// TwinCAT 3 PLC project AngerbauerWilhelm
// ProgramVersion: 3.1.4023.0
// libraries:
//   EfficientIO Communicator, * (EfficientIO)
//   EfficientIO Energy Basic, * (EfficientIO)
//   EfficientIO ModbusTCP, * (EfficientIO)
//   Lynus Persistent Data V1, * (Lynus AG)
//   Lynus Standards, * (EfficientIO)
//   Tc2_Standard, * (Beckhoff Automation GmbH)
//   Tc2_System, * (Beckhoff Automation GmbH)
//   Tc2_TcpIp, * (Beckhoff Automation GmbH)
//   Tc2_Utilities, * (Beckhoff Automation GmbH)
//   Tc3_Module, * (Beckhoff Automation GmbH)
// project tree:
//   / FastTask.TcTTO, PlcTask.TcTTO, SlowTask.TcTTO
//   FBs/ fb_Convert4BytesToLreal.TcPOU (not stored), FB_ModBus_100Registers_FC3.TcPOU, FB_ModBus_2Registers_FC3.TcPOU (not stored), FB_TCPModbusRequest_PV.TcPOU, FB_TCPModbusRequest_Grid.TcPOU
//   POUs/ prgComEffIO.TcPOU, prgGrid.TcPOU, prgPersistent.TcPOU (not stored), prgPV.TcPOU, prgRWEffIO.TcPOU, prgTCP.TcPOU, prgVarEffIO.TcPOU
// real-time tasks:
//   TASK MiddleTask: cycle T#10ms, priority 20, ADS port 350
//   TASK FastTask: cycle T#5ms, priority 19, ADS port 351
//   TASK SlowTask: cycle T#20ms, priority 21, ADS port 352

CONFIGURATION AngerbauerWilhelm
    RESOURCE PLC ON TwinCAT3
        TASK FastTask(INTERVAL := T#5ms, PRIORITY := 19);
        TASK PlcTask(INTERVAL := T#10ms, PRIORITY := 20);
        TASK SlowTask(INTERVAL := T#20ms, PRIORITY := 21);
        PROGRAM prgRWEffIO WITH FastTask : prgRWEffIO;
        PROGRAM prgVarEffIO WITH FastTask : prgVarEffIO;
        PROGRAM prgTCP WITH PlcTask : prgTCP;
        PROGRAM prgPV WITH PlcTask : prgPV;
        PROGRAM prgPersistent WITH PlcTask : prgPersistent;
        PROGRAM prgGrid WITH PlcTask : prgGrid;
        PROGRAM prgComEffIO WITH SlowTask : prgComEffIO;
    END_RESOURCE
END_CONFIGURATION

// ---- POUs/prgRWEffIO.TcPOU
PROGRAM prgRWEffIO
VAR
	fbRW1		: FB_ReadWrite_V2;
END_VAR

fbRW1(eUploadType:=	eSelectDataUploadType.e_Change_Intervall5min, 
					bBusy=> , 
					bError=> , 
					udiErrorCodeOut=> , 
					eErrorReadWrite_Out=> );

END_PROGRAM

// ---- POUs/prgVarEffIO.TcPOU
PROGRAM prgVarEffIO
VAR
	fbVar		: FB_VarInfo;
END_VAR

fbVar(
	bReadInfo:= , 
	eTMCFile:= eSelectTMCFile.eDontUseTMCFile, 
	eSavePositionTMCFile:= eSavePositionOnPLC.ePostionC, 
	udiCounterFoundVariables=> , 
	bError=> , 
	bBusy=> , 
	byProgress=> , 
	udiErrorCodeOut=> , 
	eErrorVarInfo_Out=> , 
	sVarWithError=> );

END_PROGRAM

// ---- POUs/prgTCP.TcPOU
PROGRAM prgTCP
VAR
	FB_SocketConnect : FB_SocketConnect;
	bExecuteSC: BOOL;
	hSocket : T_HSOCKET;
	FB_SocketSend : FB_SocketSend;
	sSendString : STRING(255);
	byteSendString : ARRAY[1..12] OF BYTE;
	bExecuteSS: BOOL;
	FB_SocketReceive : FB_SocketReceive;
	byteReceiveString : ARRAY[1..200] OF BYTE;
	FB_BYTE_TO_WORD : FB_CV_BYTE_TO_WORD;
	FB_WORD_TO_INT : FB_CV_WORD_TO_INT;
	wTemp : WORD;
	iOutput : INT;

END_VAR

FB_SocketConnect(
	sSrvNetId := '',
	sRemoteHost := '10.0.0.4',
	nRemotePort := 502,
	bExecute := bExecuteSC,
	tTimeout := T#1S,
	bBusy =>,
	bError =>,
	nErrId =>,
	hSocket => hSocket);
	
FB_SocketSend(
	sSrvNetId:= '', 
	hSocket:= hSocket, 
	cbLen:= 12,
	pSrc:= ADR( byteSendString ), 
	bExecute:= bExecuteSS, 
	tTimeout:= T#3S, 
	bBusy=> , 
	bError=> , 
	nErrId=> );

FB_SocketReceive(
	sSrvNetId:= '', 
	hSocket:= hSocket, 
	cbLen:= 200, 
	pDest:= ADR( byteReceiveString ), 
	bExecute:= , 
	tTimeout:= T#3S, 
	bBusy=> , 
	bError=> , 
	nErrId=> , 
	nRecBytes=> );
	
FB_BYTE_TO_WORD(byInputValue_1 := byteReceiveString[12],byInputValue_2 := byteReceiveString[13], Ebyteorderforconvert := Ebyteorder.EBIGENDIAN, woutputvalue => wTemp);
FB_WORD_TO_INT(wInputValue := wTemp, iOutputValue => iOutput);

END_PROGRAM

// ---- POUs/prgPV.TcPOU
PROGRAM prgPV
VAR
	fbPVCounter1		: FB_EnergyCounter;
	fbPVCounter2		: FB_EnergyCounter;
	lrPowerPV1			: LREAL;				//{#lynus.ag#()}
	lrPowerPV2			: LREAL;				//{#lynus.ag#()}
	lrPowerPVTotal		: LREAL;				//{#lynus.ag#()}
	byErrorWarningPV	: BYTE;					//{#lynus.ag#()}
	FB_PV1:FB_TCPModbusRequest_PV;
	FB_PV2:FB_TCPModbusRequest_PV;
	lrVoltagePV1_L1L2_V		: LREAL;				//{#lynus.ag#()}
	lrVoltagePV1_L2L3_V		: LREAL;				//{#lynus.ag#()}
	lrVoltagePV1_L3L1_V		: LREAL;				//{#lynus.ag#()}
	lrVoltagePV2_L1L2_V		: LREAL;				//{#lynus.ag#()}
	lrVoltagePV2_L2L3_V		: LREAL;				//{#lynus.ag#()}
	lrVoltagePV2_L3L1_V		: LREAL;				//{#lynus.ag#()}
END_VAR
VAR PERSISTENT
	lrCounterPV1		: LREAL;					//{#lynus.ag#()}
	lrCounterPV2		: LREAL;					//{#lynus.ag#()}
	lrCounterPVTotal	: LREAL;					//{#lynus.ag#()}
END_VAR


FB_PV1	(	b_Enable:= TRUE, 
			str_IPAdress:= '10.0.0.4', 
			lreal_RealPower_kW=> lrPowerPV1,
			lreal_Voltage_L1L2_V=> lrVoltagePV1_L1L2_V , 
			lreal_Voltage_L2L3_V=> lrVoltagePV1_L2L3_V , 
			lreal_Voltage_L3L1_V=> lrVoltagePV1_L3L1_V);


fbPVCounter1(	byActiveTariff := 1,	
				lrPowerInput := 0-lrPowerPV1,
				lrTotalCounterEnergy_Production => lrCounterPV1);
	

FB_PV2	(	b_Enable:= TRUE, 
			str_IPAdress:= '10.0.0.5', 
			lreal_RealPower_kW=> lrPowerPV2,
			lreal_Voltage_L1L2_V=> lrVoltagePV2_L1L2_V , 
			lreal_Voltage_L2L3_V=> lrVoltagePV2_L2L3_V , 
			lreal_Voltage_L3L1_V=> lrVoltagePV2_L3L1_V);

fbPVCounter2(	byActiveTariff := 1,	
				lrPowerInput := 0-lrPowerPV2,
				lrTotalCounterEnergy_Production => lrCounterPV2);
	
lrPowerPVTotal := lrPowerPV1 + lrPowerPV2;
lrCounterPVTotal := lrCounterPV1 + lrCounterPV2;

END_PROGRAM

// ---- FBs/FB_TCPModbusRequest_PV.TcPOU
FUNCTION_BLOCK FB_TCPModbusRequest_PV
VAR_INPUT
	b_Enable: BOOL;
	str_IPAdress: STRING(15);
	
		
END_VAR
VAR_OUTPUT

	lreal_RealPower_kW:LREAL;
	lreal_Voltage_L1L2_V: LREAL;
	lreal_Voltage_L2L3_V: LREAL;
	lreal_Voltage_L3L1_V: LREAL;
	lreal_Voltage_L1_V: LREAL;
	lreal_Voltage_L2_V: LREAL;
	lreal_Voltage_L3_V: LREAL;
	lreal_Current_L1_A: LREAL;
	lreal_Current_L2_A: LREAL;
	lreal_Current_L3_A: LREAL;
	lreal_PeakPowerDay_kW: LREAL;
	lreal_Power2_kW: LREAL;
	lreal_ReactivePower_kVAr: LREAL;
	lreal_PowerFactor: LREAL;
	lreal_Frequency_Hz: LREAL;
	lreal_Efficiency: LREAL;
	lreal_InternalTemperature_C: LREAL;
	lreal_IsolationResistance_MOhm: LREAL;
END_VAR
VAR
	i_State:INT;
	FB_SocketConnect : FB_SocketConnect;
	hSocket : T_HSOCKET;
	FB_SocketSend : FB_SocketSend;
	FB_SocketReceive : FB_SocketReceive;
	byteSendString : ARRAY[1..12] OF BYTE;
	FB_CloseSockets: FB_SocketCloseAll;
	
	ton_TimeOut: Ton;
	ton_WaitforReconnect: Ton;
	ton_ConnectionEstablised: Ton;
	time_ReconnectTime:TIME:=T#30M;
	b_configured: BOOL;
	byteReceiveString : ARRAY[1..200] OF BYTE;
	FB_BYTE_TO_WORD_1 : FB_CV_BYTE_TO_WORD;
	FB_BYTE_TO_WORD_2 : FB_CV_BYTE_TO_WORD;
	FB_WORD_TO_INT : FB_CV_WORD_TO_INT;
	ton_WaitforNetxtRequest: Ton;
	ton_Wait: Ton;
	int_SuccessCounter: INT;
	int_ReconnectCounter: INT;
	int_ErrorCount: INT;
	fbConvertWordToDword		: FB_CV_WORD_TO_DWORD;			//Convert Word to Dword
	fb_ConvertBytesToLreal		:fb_Convert4BytesToLreal;

END_VAR





IF NOT b_Enable THEN			// go to state 0 if not enabled
	i_State := 0;
END_IF


CASE i_State OF
	0:	// wait for enable state
		IF b_Enable THEN
			i_State := 1;
		END_IF
		FB_SocketConnect.bExecute := FALSE;
		FB_SocketSend.bExecute := FALSE;
		FB_SocketSend.bExecute := FALSE;
		ton_TimeOut.IN :=FALSE;	
		ton_ConnectionEstablised.IN := FALSE;
	

	1: // check if configured
		IF b_configured = FALSE THEN
			// request FC3, Register 32064, 25 Words --> Real PV Power ff
			byteSendString[1] := 0;
			byteSendString[2] := 1;
			byteSendString[3] := 0;
			byteSendString[4] := 0;
			byteSendString[5] := 0;
			byteSendString[6] := 6;
			byteSendString[7] := 1;
			byteSendString[8] := 3;
			byteSendString[9] := 125;
			byteSendString[10] := 64;
			byteSendString[11] := 0;
			byteSendString[12] := 25;
		
			b_configured := TRUE;
		END_IF
		i_State := i_State+1;
		
	2: // open socket
		FB_SocketConnect.bExecute := TRUE;
		ton_TimeOut.IN :=TRUE;
		i_State := i_State+1;
		
	3: // wait for connection established	
		IF NOT FB_SocketConnect.bBusy AND NOT FB_SocketConnect.bError THEN
			ton_TimeOut.IN :=FALSE;
			ton_ConnectionEstablised.IN := TRUE;
			i_State := i_State+1;
		ELSIF FB_SocketConnect.bError OR ton_TimeOut.Q THEN
			ton_TimeOut.IN :=FALSE;
			i_State := 100;
		END_IF
	
	4: //connection established, request data
		ton_Wait.IN := TRUE;
		IF ton_Wait.Q THEN
			FB_SocketSend.bExecute := TRUE;
			ton_TimeOut.IN :=TRUE;
			ton_Wait.IN := FALSE;
			i_State := i_State+1;
		END_IF
	
	5: // wait for request sent
		IF NOT FB_SocketSend.bBusy AND NOT FB_SocketSend.bError THEN
			ton_TimeOut.IN :=FALSE;
			FB_SocketSend.bExecute := FALSE;
			i_State := i_State+1;  
		ELSIF FB_SocketSend.bError OR ton_TimeOut.Q THEN
			FB_SocketSend.bExecute := FALSE;
			ton_TimeOut.IN :=FALSE;
			i_State := 100;
		END_IF
		
	6: // wait for data
		ton_Wait.IN := TRUE;
		IF ton_Wait.Q THEN
			FB_SocketReceive.bExecute := TRUE;
			ton_Wait.IN := FALSE;
			i_State := i_State+1; 
		END_IF		 
	
	7:	
		ton_Wait.IN := TRUE;
		IF ton_Wait.Q THEN
			ton_TimeOut.IN :=TRUE;
			i_State := i_State+1; 
		END_IF	
	
	8: // convert received data
		IF NOT FB_SocketReceive.bBusy AND NOT FB_SocketReceive.bError THEN
			int_SuccessCounter := int_SuccessCounter+1;
			ton_TimeOut.IN :=FALSE;
			FB_SocketReceive.bExecute := FALSE;
	
			FB_BYTE_TO_WORD_1(byInputValue_1 := byteReceiveString[14],byInputValue_2 := byteReceiveString[15], Ebyteorderforconvert := Ebyteorder.EBIGENDIAN, woutputvalue => );
			lreal_Voltage_L1L2_V := WORD_TO_LREAL(FB_BYTE_TO_WORD_1.woutputvalue)/10;
			FB_BYTE_TO_WORD_1(byInputValue_1 := byteReceiveString[16],byInputValue_2 := byteReceiveString[17], Ebyteorderforconvert := Ebyteorder.EBIGENDIAN, woutputvalue => );
			lreal_Voltage_L2L3_V := WORD_TO_LREAL(FB_BYTE_TO_WORD_1.woutputvalue)/10;
			FB_BYTE_TO_WORD_1(byInputValue_1 := byteReceiveString[18],byInputValue_2 := byteReceiveString[19], Ebyteorderforconvert := Ebyteorder.EBIGENDIAN, woutputvalue => );
			lreal_Voltage_L3L1_V := WORD_TO_LREAL(FB_BYTE_TO_WORD_1.woutputvalue)/10;
			FB_BYTE_TO_WORD_1(byInputValue_1 := byteReceiveString[20],byInputValue_2 := byteReceiveString[21], Ebyteorderforconvert := Ebyteorder.EBIGENDIAN, woutputvalue => );
			lreal_Voltage_L1_V := WORD_TO_LREAL(FB_BYTE_TO_WORD_1.woutputvalue)/10;
			FB_BYTE_TO_WORD_1(byInputValue_1 := byteReceiveString[22],byInputValue_2 := byteReceiveString[23], Ebyteorderforconvert := Ebyteorder.EBIGENDIAN, woutputvalue => );
			lreal_Voltage_L2_V := WORD_TO_LREAL(FB_BYTE_TO_WORD_1.woutputvalue)/10;
			FB_BYTE_TO_WORD_1(byInputValue_1 := byteReceiveString[24],byInputValue_2 := byteReceiveString[25], Ebyteorderforconvert := Ebyteorder.EBIGENDIAN, woutputvalue => );
			lreal_Voltage_L3_V := WORD_TO_LREAL(FB_BYTE_TO_WORD_1.woutputvalue)/10;


			fb_ConvertBytesToLreal(	by_InputValue_1:= byteReceiveString[10], 
									by_InputValue_2:= byteReceiveString[11], 
									by_InputValue_3:= byteReceiveString[12], 
									by_InputValue_4:= byteReceiveString[13], 
									int_Divider:= 1000, 
									lreal_Output=> );

			IF fb_ConvertBytesToLreal.lreal_Output < 30 AND fb_ConvertBytesToLreal.lreal_Output > -1 THEN
				lreal_RealPower_kW := fb_ConvertBytesToLreal.lreal_Output;
			END_IF
			
			fb_ConvertBytesToLreal(	by_InputValue_1:= byteReceiveString[26], 
									by_InputValue_2:= byteReceiveString[27], 
									by_InputValue_3:= byteReceiveString[28], 
									by_InputValue_4:= byteReceiveString[29], 
									int_Divider:= 1000, 
									lreal_Output=> lreal_Current_L1_A);
									
			fb_ConvertBytesToLreal(	by_InputValue_1:= byteReceiveString[30], 
									by_InputValue_2:= byteReceiveString[31], 
									by_InputValue_3:= byteReceiveString[32], 
									by_InputValue_4:= byteReceiveString[33], 
									int_Divider:= 1000, 
									lreal_Output=> lreal_Current_L2_A);

			fb_ConvertBytesToLreal(	by_InputValue_1:= byteReceiveString[34], 
									by_InputValue_2:= byteReceiveString[35], 
									by_InputValue_3:= byteReceiveString[36], 
									by_InputValue_4:= byteReceiveString[37], 
									int_Divider:= 1000, 
									lreal_Output=> lreal_Current_L3_A);
									
			fb_ConvertBytesToLreal(	by_InputValue_1:= byteReceiveString[38], 
									by_InputValue_2:= byteReceiveString[39], 
									by_InputValue_3:= byteReceiveString[40], 
									by_InputValue_4:= byteReceiveString[41], 
									int_Divider:= 1000, 
									lreal_Output=> lreal_PeakPowerDay_kW );

			fb_ConvertBytesToLreal(	by_InputValue_1:= byteReceiveString[42], 
									by_InputValue_2:= byteReceiveString[43], 
									by_InputValue_3:= byteReceiveString[44], 
									by_InputValue_4:= byteReceiveString[45], 
									int_Divider:= 1000, 
									lreal_Output=> lreal_Power2_kW);
			
			fb_ConvertBytesToLreal(	by_InputValue_1:= byteReceiveString[46], 
									by_InputValue_2:= byteReceiveString[47], 
									by_InputValue_3:= byteReceiveString[48], 
									by_InputValue_4:= byteReceiveString[49], 
									int_Divider:= 1000, 
									lreal_Output=>lreal_ReactivePower_kVAr );

			FB_BYTE_TO_WORD_1(byInputValue_1 := byteReceiveString[50],byInputValue_2 := byteReceiveString[51], Ebyteorderforconvert := Ebyteorder.EBIGENDIAN, woutputvalue => );
			lreal_PowerFactor := WORD_TO_LREAL(FB_BYTE_TO_WORD_1.woutputvalue)/1000;
			FB_BYTE_TO_WORD_1(byInputValue_1 := byteReceiveString[52],byInputValue_2 := byteReceiveString[53], Ebyteorderforconvert := Ebyteorder.EBIGENDIAN, woutputvalue => );
			lreal_Frequency_Hz := WORD_TO_LREAL(FB_BYTE_TO_WORD_1.woutputvalue)/100;
			FB_BYTE_TO_WORD_1(byInputValue_1 := byteReceiveString[54],byInputValue_2 := byteReceiveString[55], Ebyteorderforconvert := Ebyteorder.EBIGENDIAN, woutputvalue => );
			lreal_Efficiency := WORD_TO_LREAL(FB_BYTE_TO_WORD_1.woutputvalue)/100;
			FB_BYTE_TO_WORD_1(byInputValue_1 := byteReceiveString[56],byInputValue_2 := byteReceiveString[57], Ebyteorderforconvert := Ebyteorder.EBIGENDIAN, woutputvalue => );
			lreal_InternalTemperature_C := WORD_TO_LREAL(FB_BYTE_TO_WORD_1.woutputvalue)/10;
			FB_BYTE_TO_WORD_1(byInputValue_1 := byteReceiveString[58],byInputValue_2 := byteReceiveString[59], Ebyteorderforconvert := Ebyteorder.EBIGENDIAN, woutputvalue => );
			lreal_IsolationResistance_MOhm := WORD_TO_LREAL(FB_BYTE_TO_WORD_1.woutputvalue)/1000;

		
			//FB_WORD_TO_INT(wInputValue := FB_BYTE_TO_WORD.woutputvalue, iOutputValue => );
			//lreal_RealPower_kW := (INT_TO_LREAL(FB_WORD_TO_INT.iOutputValue))/1000;

			i_State := i_State+1;
		ELSIF FB_SocketSend.bError OR ton_TimeOut.Q THEN
 			FB_SocketReceive.bExecute := FALSE;
			ton_TimeOut.IN :=FALSE;
			i_State := 100;
		END_IF
	
	9: // for for next request
		ton_WaitforNetxtRequest.IN := TRUE;
		IF NOT b_Enable THEN
			ton_WaitforNetxtRequest.IN := FALSE;
			i_State := 10;
		END_IF
		IF ton_WaitforNetxtRequest.Q THEN
			ton_WaitforNetxtRequest.IN := FALSE;
			i_State := 4;
		END_IF
		IF 	ton_ConnectionEstablised.Q THEN 
			ton_WaitforNetxtRequest.IN := FALSE;
			i_State := 10;
		END_IF

	10: // close sockets
		FB_CloseSockets.bExecute := TRUE;
		ton_TimeOut.IN :=TRUE;
		i_State := i_State+1;
		
	11: // wait for sockets closed
		
		IF NOT FB_CloseSockets.bBusy THEN
			int_ReconnectCounter := int_ReconnectCounter+1;
			FB_CloseSockets.bExecute := FALSE;
			i_State := 0;
		ELSIF FB_CloseSockets.bError THEN
			int_ReconnectCounter := int_ReconnectCounter+1;
			FB_CloseSockets.bExecute := FALSE;
			i_State := 0;
		END_IF

	100: // wait state for reconect
		
		FB_SocketConnect.bExecute := FALSE;
		FB_SocketSend.bExecute := FALSE;
		FB_SocketReceive.bExecute := FALSE;
		ton_ConnectionEstablised.IN := FALSE;
		ton_TimeOut.IN :=FALSE;
		ton_WaitforReconnect.IN := TRUE;
		IF ton_WaitforReconnect.Q THEN
			int_ErrorCount := int_ErrorCount+1;
			ton_WaitforReconnect.IN := FALSE;
			i_State := 10;
		END_IF
	
END_CASE



FB_SocketConnect(
	sSrvNetId := '',
	sRemoteHost := str_IPAdress,
	nRemotePort := 502,
	bExecute := ,
	tTimeout := T#1S,
	bBusy =>,
	bError =>,
	nErrId =>,
	hSocket => hSocket);
	
FB_SocketSend(
	sSrvNetId:= '', 
	hSocket:= hSocket, 
	cbLen:= 12,
	pSrc:= ADR( byteSendString ), 
	bExecute:= , 
	tTimeout:= T#3S, 
	bBusy=> , 
	bError=> , 
	nErrId=> );
	
FB_SocketReceive(
	sSrvNetId:= '', 
	hSocket:= hSocket, 
	cbLen:= 200, 
	pDest:= ADR( byteReceiveString ), 
	bExecute:= , 
	tTimeout:= T#3S, 
	bBusy=> , 
	bError=> , 
	nErrId=> , 
	nRecBytes=> );

FB_CloseSockets(
	sSrvNetId:= '', 
	bExecute:= , 
	tTimeout:= T#2S, 
	bBusy=> , 
	bError=> , 
	nErrId=> );
	
ton_TimeOut(PT := T#5S);
ton_WaitforReconnect(PT := T#10S);
ton_ConnectionEstablised(pt := time_ReconnectTime);
ton_WaitforNetxtRequest(PT:= T#10S);
ton_Wait(PT:=T#2S);

END_FUNCTION_BLOCK

// ---- POUs/prgGrid.TcPOU
PROGRAM prgGrid
VAR
	FB_PV1:FB_TCPModbusRequest_Grid;
	FB_PV2:FB_TCPModbusRequest_Grid;

	lreal_GridVoltage_L1L2_V_PV1		: LREAL;				//{#lynus.ag#()}
	lreal_GridVoltage_L2L3_V_PV1		: LREAL;				//{#lynus.ag#()}
	lreal_GridVoltage_L3L1_V_PV1		: LREAL;				//{#lynus.ag#()}
	lreal_GridVoltage_L1_V_PV1			: LREAL;				//{#lynus.ag#()}
	lreal_GridVoltage_L2_V_PV1			: LREAL;				//{#lynus.ag#()}
	lreal_GridVoltage_L3_V_PV1			: LREAL;				//{#lynus.ag#()}
	lreal_GridCurrent_L1_A_PV1			: LREAL;				//{#lynus.ag#()}
	lreal_GridCurrent_L2_A_PV1			: LREAL;				//{#lynus.ag#()}
	lreal_GridCurrent_L3_A_PV1			: LREAL;				//{#lynus.ag#()}
	lreal_GridPower_kW_PV1				: LREAL;				//{#lynus.ag#()}
	lreal_GridPower_kW_PV1_2			: LREAL;				//{#lynus.ag#()}
	lreal_GridReactivePower_kVAr_PV1	: LREAL;				//{#lynus.ag#()}
	lreal_GridPowerFactor_PV1			: LREAL;				//{#lynus.ag#()}
	lreal_GridFrequency_Hz_PV1			: LREAL;				//{#lynus.ag#()}
	lreal_GridEnergyDelivered_kWh_PV1	: LREAL;				//{#lynus.ag#()}
	lreal_GridEnergySupllied_kWh_PV1	: LREAL;				//{#lynus.ag#()}
	
	lreal_GridVoltage_L1L2_V_PV2		: LREAL;				//{#lynus.ag#()}
	lreal_GridVoltage_L2L3_V_PV2		: LREAL;				//{#lynus.ag#()}
	lreal_GridVoltage_L3L1_V_PV2		: LREAL;				//{#lynus.ag#()}
	lreal_GridVoltage_L1_V_PV2			: LREAL;				//{#lynus.ag#()}
	lreal_GridVoltage_L2_V_PV2			: LREAL;				//{#lynus.ag#()}
	lreal_GridVoltage_L3_V_PV2			: LREAL;				//{#lynus.ag#()}
	lreal_GridCurrent_L1_A_PV2			: LREAL;				//{#lynus.ag#()}
	lreal_GridCurrent_L2_A_PV2			: LREAL;				//{#lynus.ag#()}
	lreal_GridCurrent_L3_A_PV2			: LREAL;				//{#lynus.ag#()}
	lreal_GridPower_kW_PV2				: LREAL;				//{#lynus.ag#()}
	lreal_GridPower_kW_PV2_2			: LREAL;				//{#lynus.ag#()}
	lreal_GridReactivePower_kVAr_PV2	: LREAL;				//{#lynus.ag#()}
	lreal_GridPowerFactor_PV2			: LREAL;				//{#lynus.ag#()}
	lreal_GridFrequency_Hz_PV2			: LREAL;				//{#lynus.ag#()}
	lreal_GridEnergyDelivered_kWh_PV2	: LREAL;				//{#lynus.ag#()}
	lreal_GridEnergySupllied_kWh_PV2	: LREAL;				//{#lynus.ag#()}

	lreal_HousePower_kW_PV1				: LREAL;				//{#lynus.ag#()}
	lreal_HousePower_kW_PV2				: LREAL;				//{#lynus.ag#()}
	lreal_HousePower_kW_PV1_2			: LREAL;				//{#lynus.ag#()}
	lreal_HousePower_kW_PV2_2			: LREAL;				//{#lynus.ag#()}
	
	lreal_GridPower_kW_Total			: LREAL;				//{#lynus.ag#()}

END_VAR


FB_PV1	(	b_Enable:= TRUE, 
			str_IPAdress:= prgPv.FB_PV1.str_IPAdress);


FB_PV2	(	b_Enable:= TRUE, 
			str_IPAdress:= prgPv.FB_PV2.str_IPAdress);



lreal_GridVoltage_L1L2_V_PV1 	:= FB_PV1.lreal_GridVoltage_L1L2_V;
lreal_GridVoltage_L2L3_V_PV1 	:= FB_PV1.lreal_GridVoltage_L2L3_V;
lreal_GridVoltage_L3L1_V_PV1 	:= FB_PV1.lreal_GridVoltage_L3L1_V;
lreal_GridVoltage_L1_V_PV1		:= FB_PV1.lreal_GridVoltage_L1_V;
lreal_GridVoltage_L2_V_PV1		:= FB_PV1.lreal_GridVoltage_L2_V;
lreal_GridVoltage_L3_V_PV1		:= FB_PV1.lreal_GridVoltage_L3_V;
lreal_GridCurrent_L1_A_PV1		:= FB_PV1.lreal_GridCurrent_L1_A;
lreal_GridCurrent_L2_A_PV1		:= FB_PV1.lreal_GridCurrent_L2_A;
lreal_GridCurrent_L3_A_PV1		:= FB_PV1.lreal_GridCurrent_L3_A;
lreal_GridPower_kW_PV1			:= FB_PV1.lreal_GridPower_kW;
lreal_GridPower_kW_PV1_2		:= FB_PV1.lreal_GridPower_kW * (-1);
lreal_GridReactivePower_kVAr_PV1:= FB_PV1.lreal_GridReactivePower_kVAr;
lreal_GridPowerFactor_PV1		:= FB_PV1.lreal_GridPowerFactor;
lreal_GridFrequency_Hz_PV1		:= FB_PV1.lreal_GridFrequency_Hz;
lreal_GridEnergyDelivered_kWh_PV1:= FB_PV1.lreal_GridEnergyDelivered_kWh;
lreal_GridEnergySupllied_kWh_PV1 := FB_PV1.lreal_GridEnergySupllied_kWh;

lreal_HousePower_kW_PV1 := lreal_GridPower_kW_PV1 + prgPV.lrPowerPV1;
lreal_HousePower_kW_PV1_2 := lreal_GridPower_kW_PV1_2 + prgPV.lrPowerPV1;

lreal_GridVoltage_L1L2_V_PV2 	:= FB_PV2.lreal_GridVoltage_L1L2_V;
lreal_GridVoltage_L2L3_V_PV2 	:= FB_PV2.lreal_GridVoltage_L2L3_V;
lreal_GridVoltage_L3L1_V_PV2 	:= FB_PV2.lreal_GridVoltage_L3L1_V;
lreal_GridVoltage_L1_V_PV2		:= FB_PV2.lreal_GridVoltage_L1_V;
lreal_GridVoltage_L2_V_PV2		:= FB_PV2.lreal_GridVoltage_L2_V;
lreal_GridVoltage_L3_V_PV2		:= FB_PV2.lreal_GridVoltage_L3_V;
lreal_GridCurrent_L1_A_PV2		:= FB_PV2.lreal_GridCurrent_L1_A;
lreal_GridCurrent_L2_A_PV2		:= FB_PV2.lreal_GridCurrent_L2_A;
lreal_GridCurrent_L3_A_PV2		:= FB_PV2.lreal_GridCurrent_L3_A;
lreal_GridPower_kW_PV2			:= FB_PV2.lreal_GridPower_kW;
lreal_GridPower_kW_PV2_2		:= FB_PV2.lreal_GridPower_kW * (-1);
lreal_GridReactivePower_kVAr_PV2:= FB_PV2.lreal_GridReactivePower_kVAr;
lreal_GridPowerFactor_PV2		:= FB_PV2.lreal_GridPowerFactor;
lreal_GridFrequency_Hz_PV2		:= FB_PV2.lreal_GridFrequency_Hz;
lreal_GridEnergyDelivered_kWh_PV2:= FB_PV2.lreal_GridEnergyDelivered_kWh;
lreal_GridEnergySupllied_kWh_PV2 := FB_PV2.lreal_GridEnergySupllied_kWh;


lreal_HousePower_kW_PV2 := lreal_GridPower_kW_PV2 + prgPV.lrPowerPV2;
lreal_HousePower_kW_PV2_2 := lreal_GridPower_kW_PV2_2 + prgPV.lrPowerPV2;

lreal_GridPower_kW_Total := lreal_GridPower_kW_PV1_2 + lreal_GridPower_kW_PV2_2;

END_PROGRAM

// ---- FBs/FB_TCPModbusRequest_Grid.TcPOU
FUNCTION_BLOCK FB_TCPModbusRequest_Grid
VAR_INPUT
	b_Enable: BOOL;
	str_IPAdress: STRING(15);
	
		
END_VAR
VAR_OUTPUT
	b_MeterOnline: BOOL;
	lreal_GridVoltage_L1L2_V: LREAL;
	lreal_GridVoltage_L2L3_V: LREAL;
	lreal_GridVoltage_L3L1_V: LREAL;
	lreal_GridVoltage_L1_V: LREAL;
	lreal_GridVoltage_L2_V: LREAL;
	lreal_GridVoltage_L3_V: LREAL;
	lreal_GridCurrent_L1_A: LREAL;
	lreal_GridCurrent_L2_A: LREAL;
	lreal_GridCurrent_L3_A: LREAL;
	lreal_GridPower_kW: LREAL;
	lreal_GridReactivePower_kVAr: LREAL;
	lreal_GridPowerFactor: LREAL;
	lreal_GridFrequency_Hz: LREAL;
	lreal_GridEnergyDelivered_kWh: LREAL;
	lreal_GridEnergySupllied_kWh: LREAL;
END_VAR
VAR
	i_State:INT;
	FB_SocketConnect : FB_SocketConnect;
	hSocket : T_HSOCKET;
	FB_SocketSend : FB_SocketSend;
	FB_SocketReceive : FB_SocketReceive;
	byteSendString : ARRAY[1..12] OF BYTE;
	FB_CloseSockets: FB_SocketCloseAll;
	
	ton_TimeOut: Ton;
	ton_WaitforReconnect: Ton;
	ton_ConnectionEstablised: Ton;
	time_ReconnectTime:TIME:=T#30M;
	b_configured: BOOL;
	byteReceiveString : ARRAY[1..200] OF BYTE;
	FB_BYTE_TO_WORD_1 : FB_CV_BYTE_TO_WORD;
	FB_BYTE_TO_WORD_2 : FB_CV_BYTE_TO_WORD;
	FB_WORD_TO_INT : FB_CV_WORD_TO_INT;
	ton_WaitforNetxtRequest: Ton;
	ton_Wait: Ton;
	int_SuccessCounter: INT;
	int_ReconnectCounter: INT;
	int_ErrorCount: INT;
	fbConvertWordToDword		: FB_CV_WORD_TO_DWORD;			//Convert Word to Dword
	fb_ConvertBytesToLreal		:fb_Convert4BytesToLreal;

END_VAR





IF NOT b_Enable THEN			// go to state 0 if not enabled
	i_State := 0;
END_IF


CASE i_State OF
	0:	// wait for enable state
		IF b_Enable THEN
			i_State := 1;
		END_IF
		FB_SocketConnect.bExecute := FALSE;
		FB_SocketSend.bExecute := FALSE;
		FB_SocketSend.bExecute := FALSE;
		ton_TimeOut.IN :=FALSE;	
		ton_ConnectionEstablised.IN := FALSE;
	

	1: // check if configured
		IF b_configured = FALSE THEN
			// request FC3, Register 37100 16#90EC, 38 Words 
			byteSendString[1] := 0;
			byteSendString[2] := 1;
			byteSendString[3] := 0;
			byteSendString[4] := 0;
			byteSendString[5] := 0;
			byteSendString[6] := 6;
			byteSendString[7] := 1;
			byteSendString[8] := 3;
			byteSendString[9] := 16#90;
			byteSendString[10] := 16#EC;
			byteSendString[11] := 0;
			byteSendString[12] := 38;
			b_configured := TRUE;
		END_IF
		i_State := i_State+1;
		
	2: // open socket
		FB_SocketConnect.bExecute := TRUE;
		ton_TimeOut.IN :=TRUE;
		i_State := i_State+1;
		
	3: // wait for connection established	
		IF NOT FB_SocketConnect.bBusy AND NOT FB_SocketConnect.bError THEN
			ton_TimeOut.IN :=FALSE;
			ton_ConnectionEstablised.IN := TRUE;
			i_State := i_State+1;
		ELSIF FB_SocketConnect.bError OR ton_TimeOut.Q THEN
			ton_TimeOut.IN :=FALSE;
			i_State := 100;
		END_IF
	
	4: //connection established, request data
		ton_Wait.IN := TRUE;
		IF ton_Wait.Q THEN
			FB_SocketSend.bExecute := TRUE;
			ton_TimeOut.IN :=TRUE;
			ton_Wait.IN := FALSE;
			i_State := i_State+1;
		END_IF
	
	5: // wait for request sent
		IF NOT FB_SocketSend.bBusy AND NOT FB_SocketSend.bError THEN
			ton_TimeOut.IN :=FALSE;
			FB_SocketSend.bExecute := FALSE;
			i_State := i_State+1;  
		ELSIF FB_SocketSend.bError OR ton_TimeOut.Q THEN
			FB_SocketSend.bExecute := FALSE;
			ton_TimeOut.IN :=FALSE;
			i_State := 100;
		END_IF
		
	6: // wait for data
		ton_Wait.IN := TRUE;
		IF ton_Wait.Q THEN
			FB_SocketReceive.bExecute := TRUE;
			ton_Wait.IN := FALSE;
			i_State := i_State+1; 
		END_IF		 
	
	7:	
		ton_Wait.IN := TRUE;
		IF ton_Wait.Q THEN
			ton_TimeOut.IN :=TRUE;
			i_State := i_State+1; 
		END_IF	
	
	8: // convert received data
		IF NOT FB_SocketReceive.bBusy AND NOT FB_SocketReceive.bError THEN
			int_SuccessCounter := int_SuccessCounter+1;
			ton_TimeOut.IN :=FALSE;
			FB_SocketReceive.bExecute := FALSE;
	
			FB_BYTE_TO_WORD_1(byInputValue_1 := byteReceiveString[10],byInputValue_2 := byteReceiveString[11], Ebyteorderforconvert := Ebyteorder.EBIGENDIAN, woutputvalue => );
			IF WORD_TO_LREAL(FB_BYTE_TO_WORD_1.woutputvalue) = 0 THEN
				b_MeterOnline :=FALSE;
			ELSIF WORD_TO_LREAL(FB_BYTE_TO_WORD_1.woutputvalue) = 1 THEN
				b_MeterOnline :=TRUE;
			END_IF
			
			fb_ConvertBytesToLreal(	by_InputValue_1:= byteReceiveString[12], 
									by_InputValue_2:= byteReceiveString[13], 
									by_InputValue_3:= byteReceiveString[14], 
									by_InputValue_4:= byteReceiveString[15], 
									int_Divider:= 10, 
									lreal_Output=> lreal_GridVoltage_L1_V );
									
			fb_ConvertBytesToLreal(	by_InputValue_1:= byteReceiveString[16], 
									by_InputValue_2:= byteReceiveString[17], 
									by_InputValue_3:= byteReceiveString[18], 
									by_InputValue_4:= byteReceiveString[19], 
									int_Divider:= 10, 
									lreal_Output=> lreal_GridVoltage_L2_V);
									
			fb_ConvertBytesToLreal(	by_InputValue_1:= byteReceiveString[20], 
									by_InputValue_2:= byteReceiveString[21], 
									by_InputValue_3:= byteReceiveString[22], 
									by_InputValue_4:= byteReceiveString[23], 
									int_Divider:= 10, 
									lreal_Output=> lreal_GridVoltage_L3_V);
								
			fb_ConvertBytesToLreal(	by_InputValue_1:= byteReceiveString[24], 
									by_InputValue_2:= byteReceiveString[25], 
									by_InputValue_3:= byteReceiveString[26], 
									by_InputValue_4:= byteReceiveString[27], 
									int_Divider:= 100, 
									lreal_Output=> lreal_GridCurrent_L1_A );
									
			fb_ConvertBytesToLreal(	by_InputValue_1:= byteReceiveString[24], 
									by_InputValue_2:= byteReceiveString[25], 
									by_InputValue_3:= byteReceiveString[26], 
									by_InputValue_4:= byteReceiveString[27], 
									int_Divider:= 100, 
									lreal_Output=> lreal_GridCurrent_L1_A );
									
			fb_ConvertBytesToLreal(	by_InputValue_1:= byteReceiveString[28], 
									by_InputValue_2:= byteReceiveString[29], 
									by_InputValue_3:= byteReceiveString[30], 
									by_InputValue_4:= byteReceiveString[31], 
									int_Divider:= 100, 
									lreal_Output=> lreal_GridCurrent_L2_A );
									
			fb_ConvertBytesToLreal(	by_InputValue_1:= byteReceiveString[32], 
									by_InputValue_2:= byteReceiveString[33], 
									by_InputValue_3:= byteReceiveString[34], 
									by_InputValue_4:= byteReceiveString[35], 
									int_Divider:= 100, 
									lreal_Output=> lreal_GridCurrent_L3_A );
									
			fb_ConvertBytesToLreal(	by_InputValue_1:= byteReceiveString[36], 
									by_InputValue_2:= byteReceiveString[37], 
									by_InputValue_3:= byteReceiveString[38], 
									by_InputValue_4:= byteReceiveString[39], 
									int_Divider:= 1000, 
									lreal_Output=> );
			
			IF fb_ConvertBytesToLreal.lreal_Output < 30 AND fb_ConvertBytesToLreal.lreal_Output > -30 THEN
				lreal_GridPower_kW := fb_ConvertBytesToLreal.lreal_Output;
			END_IF
													
			fb_ConvertBytesToLreal(	by_InputValue_1:= byteReceiveString[40], 
									by_InputValue_2:= byteReceiveString[41], 
									by_InputValue_3:= byteReceiveString[42], 
									by_InputValue_4:= byteReceiveString[43], 
									int_Divider:= 1000, 
									lreal_Output=> lreal_GridReactivePower_kVAr);
											
			//FB_BYTE_TO_WORD_1(byInputValue_1 := byteReceiveString[44],byInputValue_2 := byteReceiveString[45], Ebyteorderforconvert := Ebyteorder.EbigENDIAN, woutputvalue => );
			//lreal_GridPowerFactor := WORD_TO_LREAL(FB_BYTE_TO_WORD_1.woutputvalue)/1000;

			lreal_GridPowerFactor := INT_TO_LREAL(WORD_TO_INT((SHL(BYTE_TO_WORD(byteReceiveString[44]),8) + BYTE_TO_WORD(byteReceiveString[45]))))/1000;


		
			FB_BYTE_TO_WORD_1(byInputValue_1 := byteReceiveString[46],byInputValue_2 := byteReceiveString[47], Ebyteorderforconvert := Ebyteorder.EbigENDIAN, woutputvalue => );
			lreal_GridFrequency_Hz := WORD_TO_LREAL(FB_BYTE_TO_WORD_1.woutputvalue)/100;
			
			fb_ConvertBytesToLreal(	by_InputValue_1:= byteReceiveString[48], 
									by_InputValue_2:= byteReceiveString[49], 
									by_InputValue_3:= byteReceiveString[50], 
									by_InputValue_4:= byteReceiveString[51], 
									int_Divider:= 100, 
									lreal_Output=> lreal_GridEnergyDelivered_kWh);
									
			fb_ConvertBytesToLreal(	by_InputValue_1:= byteReceiveString[52], 
									by_InputValue_2:= byteReceiveString[53], 
									by_InputValue_3:= byteReceiveString[54], 
									by_InputValue_4:= byteReceiveString[55], 
									int_Divider:= 100, 
									lreal_Output=> lreal_GridEnergySupllied_kWh );
			
			fb_ConvertBytesToLreal(	by_InputValue_1:= byteReceiveString[62], 
									by_InputValue_2:= byteReceiveString[63], 
									by_InputValue_3:= byteReceiveString[64], 
									by_InputValue_4:= byteReceiveString[65], 
									int_Divider:= 10 , 
									lreal_Output=> lreal_GridVoltage_L1L2_V);

			fb_ConvertBytesToLreal(	by_InputValue_1:= byteReceiveString[66], 
									by_InputValue_2:= byteReceiveString[67], 
									by_InputValue_3:= byteReceiveString[68], 
									by_InputValue_4:= byteReceiveString[69], 
									int_Divider:= 10 , 
									lreal_Output=> lreal_GridVoltage_L2L3_V);

			fb_ConvertBytesToLreal(	by_InputValue_1:= byteReceiveString[70], 
									by_InputValue_2:= byteReceiveString[71], 
									by_InputValue_3:= byteReceiveString[72], 
									by_InputValue_4:= byteReceiveString[73], 
									int_Divider:= 10 , 
									lreal_Output=> lreal_GridVoltage_L3L1_V);

			i_State := i_State+1;
		ELSIF FB_SocketSend.bError OR ton_TimeOut.Q THEN
 			FB_SocketReceive.bExecute := FALSE;
			ton_TimeOut.IN :=FALSE;
			i_State := 100;
		END_IF
	
	9: // for for next request
		ton_WaitforNetxtRequest.IN := TRUE;
		IF NOT b_Enable THEN
			ton_WaitforNetxtRequest.IN := FALSE;
			i_State := 10;
		END_IF
		IF ton_WaitforNetxtRequest.Q THEN
			ton_WaitforNetxtRequest.IN := FALSE;
			i_State := 4;
		END_IF
		IF 	ton_ConnectionEstablised.Q THEN 
			ton_WaitforNetxtRequest.IN := FALSE;
			i_State := 10;
		END_IF

	10: // close sockets
		FB_CloseSockets.bExecute := TRUE;
		ton_TimeOut.IN :=TRUE;
		i_State := i_State+1;
		
	11: // wait for sockets closed
		
		IF NOT FB_CloseSockets.bBusy THEN
			int_ReconnectCounter := int_ReconnectCounter+1;
			FB_CloseSockets.bExecute := FALSE;
			i_State := 0;
		ELSIF FB_CloseSockets.bError THEN
			int_ReconnectCounter := int_ReconnectCounter+1;
			FB_CloseSockets.bExecute := FALSE;
			i_State := 0;
		END_IF

	100: // wait state for reconect
		
		FB_SocketConnect.bExecute := FALSE;
		FB_SocketSend.bExecute := FALSE;
		FB_SocketReceive.bExecute := FALSE;
		ton_ConnectionEstablised.IN := FALSE;
		ton_TimeOut.IN :=FALSE;
		ton_WaitforReconnect.IN := TRUE;
		IF ton_WaitforReconnect.Q THEN
			int_ErrorCount := int_ErrorCount+1;
			ton_WaitforReconnect.IN := FALSE;
			i_State := 10;
		END_IF
	
END_CASE



FB_SocketConnect(
	sSrvNetId := '',
	sRemoteHost := str_IPAdress,
	nRemotePort := 502,
	bExecute := ,
	tTimeout := T#1S,
	bBusy =>,
	bError =>,
	nErrId =>,
	hSocket => hSocket);
	
FB_SocketSend(
	sSrvNetId:= '', 
	hSocket:= hSocket, 
	cbLen:= 12,
	pSrc:= ADR( byteSendString ), 
	bExecute:= , 
	tTimeout:= T#3S, 
	bBusy=> , 
	bError=> , 
	nErrId=> );
	
FB_SocketReceive(
	sSrvNetId:= '', 
	hSocket:= hSocket, 
	cbLen:= 200, 
	pDest:= ADR( byteReceiveString ), 
	bExecute:= , 
	tTimeout:= T#3S, 
	bBusy=> , 
	bError=> , 
	nErrId=> , 
	nRecBytes=> );

FB_CloseSockets(
	sSrvNetId:= '', 
	bExecute:= , 
	tTimeout:= T#2S, 
	bBusy=> , 
	bError=> , 
	nErrId=> );
	
ton_TimeOut(PT := T#5S);
ton_WaitforReconnect(PT := T#10S);
ton_ConnectionEstablised(pt := time_ReconnectTime);
ton_WaitforNetxtRequest(PT:= T#10S);
ton_Wait(PT:=T#2S);

END_FUNCTION_BLOCK

// ---- POUs/prgComEffIO.TcPOU
PROGRAM prgComEffIO
VAR
	fbCom		: FB_MqttCommunicator_V5;
END_VAR

fbCom(
	bConnect:= TRUE, 
	sUserName:= '795eb4ac-ab73-423a-978c-776b62a0fa2e', 
	sUserPassword:= 'f18add2b-7af7-4562-b9b6-6e5fd1b3afa3', 
	strAuthKey:= 'ENE87365342998', 
	eSavePositionCertificate:= eSavePositionOnPLC.ePostionC, 
	bConnected=> , 
	bError=> , 
	hrErrorCode=> , 
	eConnectionState=> , 
	eErrorMessage_Out=> );

END_PROGRAM

// ---- FBs/FB_ModBus_100Registers_FC3.TcPOU
FUNCTION_BLOCK FB_ModBus_100Registers_FC3
VAR_INPUT PERSISTENT
	m_Enable					: BOOL;						//Enable the Fuctionblock and his logic
	str_IPAdress				: STRING(15);				//IP Adress of the meter
	w_Adress					: WORD;						//modbus adress
	usint_Quantity				: usINT;						//Number of Words to get polled, max 100
END_VAR
VAR_OUTPUT
	m_PollSuccessful			: BOOL;						//Poll succesfull		
	w_Array_Received			: ARRAY[1..100] OF WORD;	// received data
	udint_Error_ID				: UDINT;					// ERR ID FB_MBReadRegs
END_VAR
VAR
	
	timer_Delay					: TON;						//Timer for Delay between Requests
	
	timer_DelayStart			: TON;						//Timer to start the state machine with Delay after enabling or after the system ist restartet
	
	timer_TimeOut				: TON;						//Timer for Timeout MB Read
	
	iStateModbusRead			: INT;						//State machine for read out Data over Modbus RTU
	
	fbMBRead_FC3				: FB_MBReadRegs  ;		//Modbus Read Function (FC3)
	
	ftrig_PEnable				: f_trig;					//Internal positive Edge
	
	iStateModbusError			: INT;						//State machine for error out Data over Modbus TCP/IP	
	
	FPError_FC_3				: R_TRIG;					//Internal positive Edge
	
	arrBuffer_FC3				: ARRAY[1..100] OF WORD;		//Buffer with Data from FC3
	
	timer_Connection_ok			: TON;
	int_Data_Received			: INT;
	
	m_MBTCPError				: BOOL;
	
	int_Data_Received_old		: INT;
	
	timer_Connection_ok_TOF	: TOF;
	
	fbConvertWordToDword		: FB_CV_WORD_TO_DWORD;			//Convert Word to Dword
	
	m_Poll_ok: BOOL;
	
	timer_Wait: Ton;
	int_TimeoutError: INT;
	int_FC3Error: INT;

END_VAR

(*	{attribute 'hide'}--------------------------------------------------------------------------------------------Limits-------------------------------------------------------------------------------------*)

w_Adress := LIMIT(0,w_Adress,60000);
usint_Quantity := LIMIT(1,usint_Quantity,100);
	
(*--------------------------------------------------------------------------------------------State Machine Read--------------------------------------------------------------------------------------*)

//Timer for Delay
timer_Delay(IN:= , PT:= T#50MS, Q=> , ET=> );

//Timeout Timer is dissabled when the Init Step is aktiv or the function is not enabled
IF iStateModbusRead = 0 OR NOT m_Enable THEN 
	timer_Timeout.IN := FALSE; 
END_IF
timer_Timeout(IN:= , PT:= T#1S, Q=> , ET=> );

//Enable with Delay that not all sockets have to be created at the same time
timer_DelayStart(IN:= m_Enable, PT:= T#1S, Q=> , ET=> );
ftrig_PEnable(CLK:= timer_DelayStart.Q, Q=> );

IF ftrig_PEnable.Q AND iStateModbusRead = 0 THEN 
	iStateModbusRead := 1; 
END_IF		
		
//Not Enabled
IF NOT m_Enable THEN 
	iStateModbusRead := 0; 
	iStateModbusError := 0; 
END_IF		
		
CASE iStateModbusRead OF

	0://Init Step 
		timer_Delay.IN := FALSE;
		fbMBRead_FC3.bExecute := FALSE;
		m_Poll_ok:=FALSE;
		int_Data_Received:=0;
	
		iStateModbusRead := 1;
	
	1://read the required registers
		//Start Read
		fbMBRead_FC3.nQuantity := usint_Quantity;
		fbMBRead_FC3.nMBAddr := w_Adress;
		fbMBRead_FC3.bExecute := TRUE;
		fbMBRead_FC3.nUnitID := 1;
		timer_Timeout.IN := TRUE;
		IF fbMBRead_FC3.bBusy THEN 
			timer_Delay.IN := TRUE; 
		END_IF
		
		//Wait for Delay, copy Data and then next step
		IF NOT fbMBRead_FC3.bBusy AND NOT fbMBRead_FC3.bError AND timer_Delay.Q THEN
			m_Poll_ok:=TRUE;
			int_Data_Received:=int_Data_Received+1;
			m_MBTCPError := FALSE; 
			
			w_Array_Received := arrBuffer_FC3;
			
			
			//Go to Next Step
			timer_Timeout.IN := FALSE;
			fbMBRead_FC3.bExecute := FALSE;
			timer_Delay.IN := FALSE;		
			iStateModbusRead := 3;
		END_IF	

		//Error or Timeout
		IF FPError_FC_3.Q THEN 
			iStateModbusError := 300;
			int_FC3Error := int_FC3Error+1;
		ELSIF timer_Timeout.Q THEN  
			timer_Timeout.IN := FALSE; 	
			iStateModbusError := 300;
			int_TimeoutError := int_TimeoutError+1;
		END_IF
		
	
	3://Wait and go to step 1
		//1 because 0 is the Init Step for Read
		timer_Wait.IN := TRUE;
		
		IF timer_Wait.Q = TRUE THEN
			iStateModbusRead := 1;
			timer_Wait.IN :=FALSE;
		END_IF

			
		
		//Error on Master, changes on Inputs or Timeout
		IF timer_Timeout.Q THEN 
			iStateModbusError := 300; 
		END_IF
	
END_CASE

(* wait timer*)

timer_Wait(PT:=T#3S);


(*------------------------------------------------------------------Error and Warning----------------------------------------------------------------------------*)	
 
timer_Connection_ok			(In:=int_Data_Received<>int_Data_Received_old,PT:=T#10S);
timer_Connection_ok_TOF		(In:=NOT(int_Data_Received<>int_Data_Received_old) AND int_Data_Received>3 ,PT:=T#20S);
int_Data_Received_old:=int_Data_Received;
m_PollSuccessful:=NOT timer_Connection_ok.Q AND timer_Connection_ok_TOF.Q ;

(*------------------------------------------------------------------------------------------Modbus TCP Functions---------------------------------------------------------------------------------------------*)

fbMBRead_FC3(	sIPAddr:= str_IPAdress, 
				nTCPPort:= 502,
				cbLength:= SIZEOF(arrBuffer_FC3), 
				pDestAddr:= ADR(arrBuffer_FC3), 
				tTimeout:= T#10S,
				nErrId => udint_Error_ID);

FPError_FC_3(CLK:= fbMBRead_FC3.bError, Q=> );		

(*------------------------------------------------------------------------------------------State Machine Error---------------------------------------------------------------------------------------------*)	

CASE iStateModbusError OF
	
	300://Error
		timer_Wait.IN :=TRUE;
		timer_Delay.IN := FALSE;
		fbMBRead_FC3.bExecute := FALSE;
		m_MBTCPError := TRUE; 		
		m_Poll_ok:=FALSE;
		int_Data_Received:=0;
				//Restart from new with the Read out part after an Error
		IF timer_Wait.Q = TRUE THEN
			iStateModbusRead := 0;	
			iStateModbusError := 0;
			timer_Wait.IN :=FALSE;
			timer_Timeout.IN := FALSE;
		END_IF		
							
END_CASE

END_FUNCTION_BLOCK
